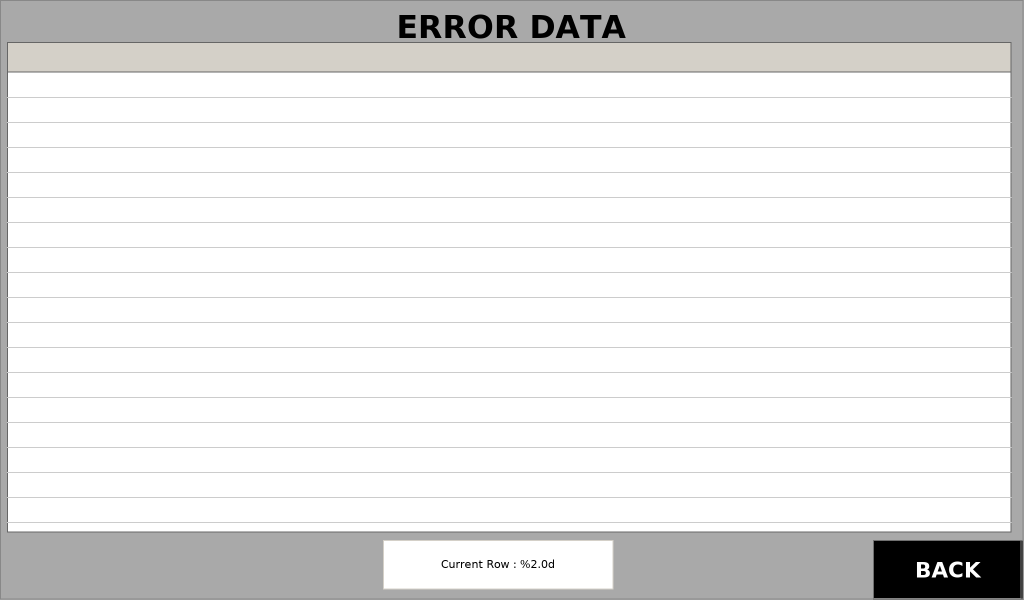
VISUALIZATION errorScreen  // 1024x600
    Label (0,10 1023x34), "ERROR DATA"
    Textfield (912,76 61x30)
    Textfield (834,76 61x30)
    Textfield (327,201 61x30)
    Textfield (555,75 84x30)
    Textfield (680,76 61x30)
    Table (7,42 1004x490), data array: GVL_machine.aErrorData
        p3854506369: GVL_machine.aErrorData[1,INDEX]
        p1892666644: GVL_machine.aErrorData[2,INDEX]
        p338671338: GVL_machine.aErrorData[3,INDEX]
        p1755163831: Function Block
        p2170511999: GVL_machine.aErrorData[4,INDEX]
        p3723444502: GVL_machine.aErrorData[5,INDEX]
        p2237128397: ERROR MESSAGE
    Button (873,540 150x60), "BACK"
        OnMouseDown: change screen: Previous maintenanceScreen3
        OnMouseDown: execute { GVL_machine.bDispErrorIcon := FALSE; }
    Textfield (383,540 230x49), "Current Row : %2.0d", text variable: GVL_machine.nErrorDataRow
END_VISUALIZATION

(* stored: Version 1.1.0.1, ProductVersion 3.1.4024.13
   Visu errorScreen: Id {27e2623b-fdf2-4371-9bbf-4ade03335c27} *)
